// TIA Portal V18 export
// export: Created 2026-06-08T16:32:20.9625212Z, ExportSetting WithDefaults, DisplayName Totally Integrated Automation Portal, DisplayVersion V18, DisplayName TIA Portal Openness, DisplayVersion V18, DisplayName TIA Portal Version Control Interface, DisplayVersion V18, DisplayName STEP 7 Professional, DisplayVersion V18, DisplayName STEP 7 Safety, DisplayVersion V18, DisplayName WinCC Professional, DisplayVersion V18
FUNCTION_BLOCK "PICK_UP_BASE_ROBOT"   // FB6, LAD
VERSION : 0.1
// stored: AutoNumber true, IsIECCheckEnabled false, UDAEnableTagReadback false
   VAR_TEMP   // added for the SCL form of the ladder/FBD networks
      _w1 : Bool;
   END_VAR
BEGIN

REGION Network 1: BASE_PICKUP_ROBOT_LOWERING_Z_AXIS
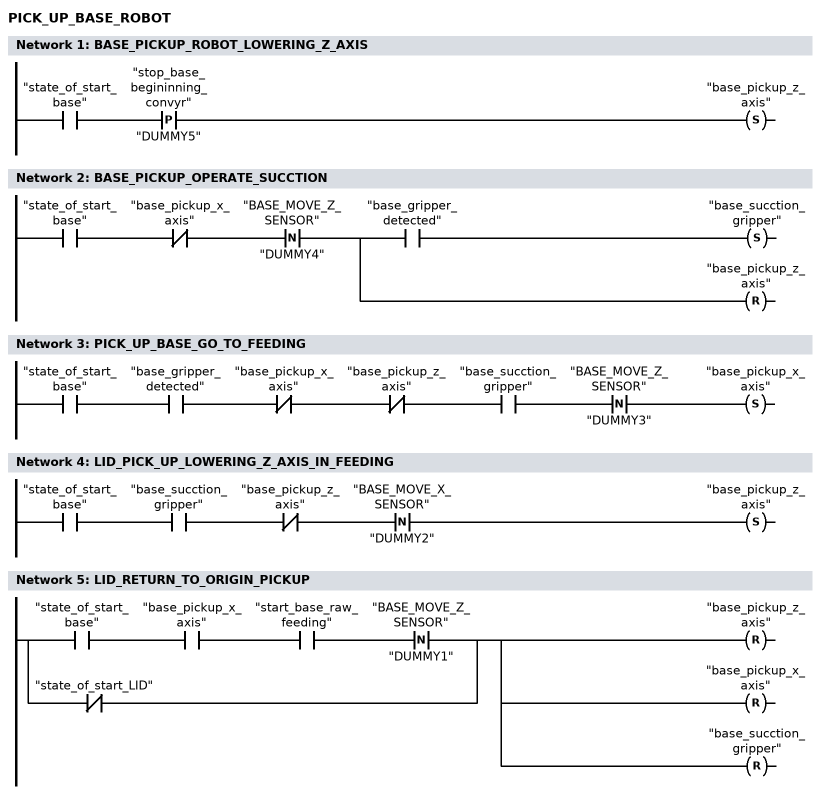
   RUNG wire#powerrail
      Contact( "state_of_start_base" )
      P_Contact(operand := "stop_base_begininning_convyr", bit := "DUMMY5")
      S_Coil( "base_pickup_z_axis" )
   END_RUNG
   // the same network as SCL:
   #_w1 := "state_of_start_base" AND "stop_base_begininning_convyr" AND NOT "DUMMY5";   // rising edge of "stop_base_begininning_convyr"
   "DUMMY5" := "stop_base_begininning_convyr";
   IF #_w1 THEN "base_pickup_z_axis" := TRUE; END_IF;
END_REGION

REGION Network 2: BASE_PICKUP_OPERATE_SUCCTION
   RUNG wire#powerrail
      Contact( "state_of_start_base" )
      I_Contact( "base_pickup_x_axis" )
      N_Contact(operand := "BASE_MOVE_Z_SENSOR", bit := "DUMMY4")
      wire#w1
      Contact( "base_gripper_detected" )
      S_Coil( "base_sucction_gripper" )
   END_RUNG
   RUNG wire#w1
      R_Coil( "base_pickup_z_axis" )
   END_RUNG
   // the same network as SCL:
   #_w1 := "state_of_start_base" AND NOT "base_pickup_x_axis" AND NOT "BASE_MOVE_Z_SENSOR" AND "DUMMY4";   // falling edge of "BASE_MOVE_Z_SENSOR"
   "DUMMY4" := "BASE_MOVE_Z_SENSOR";
   IF #_w1 AND "base_gripper_detected" THEN "base_sucction_gripper" := TRUE; END_IF;
   IF #_w1 THEN "base_pickup_z_axis" := FALSE; END_IF;
END_REGION

REGION Network 3: PICK_UP_BASE_GO_TO_FEEDING
   RUNG wire#powerrail
      Contact( "state_of_start_base" )
      Contact( "base_gripper_detected" )
      I_Contact( "base_pickup_x_axis" )
      I_Contact( "base_pickup_z_axis" )
      Contact( "base_sucction_gripper" )
      N_Contact(operand := "BASE_MOVE_Z_SENSOR", bit := "DUMMY3")
      S_Coil( "base_pickup_x_axis" )
   END_RUNG
   // the same network as SCL:
   #_w1 := "state_of_start_base" AND "base_gripper_detected" AND NOT "base_pickup_x_axis" AND NOT "base_pickup_z_axis" AND "base_sucction_gripper" AND NOT "BASE_MOVE_Z_SENSOR" AND "DUMMY3";   // falling edge of "BASE_MOVE_Z_SENSOR"
   "DUMMY3" := "BASE_MOVE_Z_SENSOR";
   IF #_w1 THEN "base_pickup_x_axis" := TRUE; END_IF;
END_REGION

REGION Network 4: LID_PICK_UP_LOWERING_Z_AXIS_IN_FEEDING
   RUNG wire#powerrail
      Contact( "state_of_start_base" )
      Contact( "base_sucction_gripper" )
      I_Contact( "base_pickup_z_axis" )
      N_Contact(operand := "BASE_MOVE_X_SENSOR", bit := "DUMMY2")
      S_Coil( "base_pickup_z_axis" )
   END_RUNG
   // the same network as SCL:
   #_w1 := "state_of_start_base" AND "base_sucction_gripper" AND NOT "base_pickup_z_axis" AND NOT "BASE_MOVE_X_SENSOR" AND "DUMMY2";   // falling edge of "BASE_MOVE_X_SENSOR"
   "DUMMY2" := "BASE_MOVE_X_SENSOR";
   IF #_w1 THEN "base_pickup_z_axis" := TRUE; END_IF;
END_REGION

REGION Network 5: LID_RETURN_TO_ORIGIN_PICKUP
   RUNG wire#powerrail
      Contact( "state_of_start_base" )
      Contact( "base_pickup_x_axis" )
      Contact( "start_base_raw_feeding" )
      N_Contact(operand := "BASE_MOVE_Z_SENSOR", bit := "DUMMY1")
      wire#w1
      R_Coil( "base_pickup_z_axis" )
   END_RUNG
   RUNG wire#powerrail
      I_Contact( "state_of_start_LID" )
   END_RUNG wire#w1
   RUNG wire#w1
      R_Coil( "base_pickup_x_axis" )
   END_RUNG
   RUNG wire#w1
      R_Coil( "base_sucction_gripper" )
   END_RUNG
   // the same network as SCL:
   #_w1 := "state_of_start_base" AND "base_pickup_x_axis" AND "start_base_raw_feeding" AND NOT "BASE_MOVE_Z_SENSOR" AND "DUMMY1";   // falling edge of "BASE_MOVE_Z_SENSOR"
   "DUMMY1" := "BASE_MOVE_Z_SENSOR";
   IF #_w1 OR NOT "state_of_start_LID" THEN
       "base_pickup_z_axis" := FALSE;
       "base_pickup_x_axis" := FALSE;
       "base_sucction_gripper" := FALSE;
   END_IF;
END_REGION
END_FUNCTION_BLOCK
